// TwinCAT 3 PLC project Rt
// Title: Rt
// Company: _
// Author: Krystian Lis et al.
// ProjectVersion: 1.0.0
// Description: Basic runtime
// ProgramVersion: 3.1.4026.9
// libraries:
//   Tc2_Standard, * (Beckhoff Automation GmbH)
//   Tc2_System, * (Beckhoff Automation GmbH)
//   Debug, * (_)
//   Results, * (_)
// project tree:
//   Runtime/Execute/ Execute.TcPOU, I_Execute.TcIO, I_ExecuteNode.TcIO
//   Runtime/ Runtime.TcPOU, _Runtime.TcGVL

// ---- Runtime/_Runtime.TcGVL
{attribute 'qualified_only'}
VAR_GLOBAL INTERNAL
	iFirstCyclic		: I_ExecuteNode;
	iLastCyclic			: I_ExecuteNode;
END_VAR

// ---- Runtime/Execute/I_Execute.TcIO
INTERFACE I_Execute EXTENDS Debug.I_Debug

METHOD Execute
VAR_INPUT
END_VAR
END_METHOD

END_INTERFACE

// ---- Runtime/Execute/I_ExecuteNode.TcIO
INTERFACE INTERNAL I_ExecuteNode EXTENDS Debug.I_Debug;

METHOD INTERNAL Attach : Results.Result
VAR_INPUT
	iExecute		: I_ExecuteNode;
END_VAR
END_METHOD

METHOD INTERNAL Exe
VAR_INPUT
END_VAR
END_METHOD

PROPERTY INTERNAL state : Results.Result
GET
END_GET
SET
END_SET
END_PROPERTY

END_INTERFACE

// ---- Runtime/Execute/Execute.TcPOU
FUNCTION_BLOCK FINAL Execute IMPLEMENTS I_ExecuteNode, Debug.I_Debug
VAR
	_iExecute		: I_Execute;
	_iNext			: I_ExecuteNode;
	_eState			: Results.Result;
END_VAR

METHOD INTERNAL Attach : Results.Result
VAR_INPUT
	iExecute		: I_ExecuteNode;
END_VAR
VAR
	_iThis			: I_ExecuteNode := THIS^;
END_VAR
IF iExecute = 0 THEN
	Debug.DebugMsg(0, Tc2_Standard.CONCAT(__POUNAME(), ': Itf = 0!'));
	RETURN;
END_IF

IF _iThis <> _Runtime.iLastCyclic THEN
	Debug.DebugMsg(THIS^, Tc2_Standard.CONCAT(__POUNAME(), ': Is not the last node!'));
	RETURN;
END_IF

IF Results.IsSome(iExecute.state) THEN
	Debug.DebugMsg(iExecute, Tc2_Standard.CONCAT(__POUNAME(), ': Has already been added!'));
	RETURN;
END_IF

_Runtime.iLastCyclic := iExecute;
_iNext := iExecute;
END_METHOD

METHOD INTERNAL Exe
VAR_INPUT
END_VAR
_iExecute.Execute();

IF _iNext <> 0 THEN
	_iNext.Exe();
END_IF
END_METHOD

//FB_Init is always available implicitly and it is used primarily for initialization.
//The return value is not evaluated. For a specific influence, you can also declare the
//methods explicitly and provide additional code there with the standard initialization
//code. You can evaluate the return value.
METHOD FB_Init: BOOL
VAR_INPUT
    bInitRetains: BOOL; // TRUE: the retain variables are initialized (reset warm / reset cold)
    bInCopyCode: BOOL;  // TRUE: the instance will be copied to the copy code afterward (online change)
	
	iExecute			: I_Execute;
END_VAR
IF Results.IsSome(_eState) THEN
	RETURN;
END_IF

IF (_iExecute := iExecute) = 0 THEN
	_eState := Results.Err.Itf0;
	Debug.DebugMsg(THIS^, Tc2_Standard.CONCAT(__POUNAME(), ': Itf = 0!'));
	RETURN;
END_IF



IF _Runtime.iLastCyclic <> 0 THEN
	IF Results.IsErr(_Runtime.iLastCyclic.Attach(THIS^), eCarry => _eState) THEN
		Debug.DebugMsg(THIS^, Tc2_Standard.CONCAT(__POUNAME(), ': Error Inside!'));
	END_IF
ELSE
	_Runtime.iFirstCyclic := THIS^;
	_Runtime.iLastCyclic := THIS^;
	_eState := Results.Ok;
END_IF
END_METHOD

PROPERTY INTERNAL state : Results.Result
GET
state := _eState;
END_GET
SET
IF Results.IsNone(_eState) THEN
	_eState := state;
END_IF
END_SET
END_PROPERTY

END_FUNCTION_BLOCK

// ---- Runtime/Runtime.TcPOU
FUNCTION Runtime

IF _Runtime.iFirstCyclic <> 0 THEN
	_Runtime.iFirstCyclic.Exe();
END_IF

END_FUNCTION
